ABB RobotStudio station: Task1.rspag

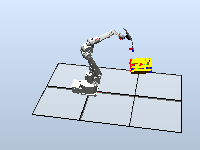
--- station ---
Station t12018 (saved by RobotStudio 6.8.8148.134)
Controller IRB_1520ID_4kg_1.50m
  mechanical unit ROB_1: IRB1520ID_4_150__02, 6 joints, base frame (0, 0, 0) mm
Layout (positions relative to the parent item):
  - IRB1520ID_4_150__02 [mechanism, from Robots\IRB1520ID_4_150_G_02.rslib] at (0, 0, 0) mm; joint values [0.6739, -0.4302, 0.2186, -0.7083, 0.9805, 0.8248] (rad or m)
  - AW_Gun_PSF_25 [mechanism, from Tools\AW_Gun_PSF_25.rslib] at (625.47, 361.2, 1236.61) mm, rotated rx -180 ry 60 rz 180 deg
  - Curve_thing [part, from Training Objects\Curve_Thing.rslib] at (900.38, 149.94, 467.04) mm, rotated rx 0 ry -5.23 rz 7.04 deg
Attachment: AW_Gun_PSF_25 is attached to IRB1520ID_4_150__02 / Link6
Targets, tools, work objects and paths stored in the station and not in the controller backup, written as RAPID:
! task T_ROB1
MODULE Module1
  CONST robtarget Target_50:=[[855.450316917,446.661091818,556.66779203],[0.05059499,0,0.998719253,0],[0,0,0,0],[9E+09,9E+09,9E+09,9E+09,9E+09,9E+09]];
  CONST robtarget Target_240:=[[870.559467167,361.195047252,567.122430983],[0.05059499,0,0.998719253,0],[0,0,0,0],[9E+09,9E+09,9E+09,9E+09,9E+09,9E+09]];
  CONST robtarget Target_60_2:=[[870.559467167,361.195047252,657.122430983],[0.05059499,0,0.998719253,0],[0,0,0,0],[9E+09,9E+09,9E+09,9E+09,9E+09,9E+09]];
  CONST robtarget Target_70_2:=[[888.080268226,219.399873941,657.122430983],[0.05059499,0,0.998719253,0],[0,0,0,0],[9E+09,9E+09,9E+09,9E+09,9E+09,9E+09]];
  CONST robtarget Target_80_2:=[[904.089387296,224.300982937,658.630621291],[0.05059499,0,0.998719253,0],[0,0,0,0],[9E+09,9E+09,9E+09,9E+09,9E+09,9E+09]];
  CONST robtarget Target_90_2:=[[920.816879189,223.596185165,660.141143018],[0.05059499,0,0.998719253,0],[0,0,0,0],[9E+09,9E+09,9E+09,9E+09,9E+09,9E+09]];
  CONST robtarget Target_100_2:=[[936.371952521,217.365147414,661.483254401],[0.05059499,0,0.998719253,0],[0,0,0,0],[9E+09,9E+09,9E+09,9E+09,9E+09,9E+09]];
  CONST robtarget Target_110_2:=[[948.996340197,206.312194788,662.505249932],[0.05059499,0,0.998719253,0],[0,0,0,0],[9E+09,9E+09,9E+09,9E+09,9E+09,9E+09]];
  CONST robtarget Target_120_2:=[[1011.676222413,214.057181596,668.281846254],[0.05059499,0,0.998719253,0],[0,0,0,0],[9E+09,9E+09,9E+09,9E+09,9E+09,9E+09]];
  CONST robtarget Target_130_2:=[[1016.694200617,232.87209655,668.948386567],[0.05059499,0,0.998719253,0],[0,0,0,0],[9E+09,9E+09,9E+09,9E+09,9E+09,9E+09]];
  CONST robtarget Target_140_2:=[[1028.495415861,248.325502176,670.192966537],[0.05059499,0,0.998719253,0],[0,0,0,0],[9E+09,9E+09,9E+09,9E+09,9E+09,9E+09]];
  CONST robtarget Target_150_2:=[[1045.287851693,258.07079632,671.826596493],[0.05059499,0,0.998719253,0],[0,0,0,0],[9E+09,9E+09,9E+09,9E+09,9E+09,9E+09]];
  CONST robtarget Target_160_2:=[[1064.521574005,260.628154485,673.601209461],[0.05059499,0,0.998719253,0],[0,0,0,0],[9E+09,9E+09,9E+09,9E+09,9E+09,9E+09]];
  CONST robtarget Target_170_2:=[[1083.275938942,255.609241416,675.247330174],[0.05059499,0,0.998719253,0],[0,0,0,0],[9E+09,9E+09,9E+09,9E+09,9E+09,9E+09]];
  CONST robtarget Target_180_2:=[[1098.703093142,243.77617988,676.514994934],[0.05059499,0,0.998719253,0],[0,0,0,0],[9E+09,9E+09,9E+09,9E+09,9E+09,9E+09]];
  CONST robtarget Target_190_2:=[[1108.460420734,226.925822191,677.211708641],[0.05059499,0,0.998719253,0],[0,0,0,0],[9E+09,9E+09,9E+09,9E+09,9E+09,9E+09]];
  CONST robtarget Target_200_2:=[[1111.06626994,207.616897902,677.231675207],[0.05059499,0,0.998719253,0],[0,0,0,0],[9E+09,9E+09,9E+09,9E+09,9E+09,9E+09]];
  CONST robtarget Target_210_2:=[[1106.124942133,188.7814703,676.571862704],[0.05059499,0,0.998719253,0],[0,0,0,0],[9E+09,9E+09,9E+09,9E+09,9E+09,9E+09]];
  CONST robtarget Target_220_2:=[[1191.583816693,199.341124094,684.447777639],[0.05059499,0,0.998719253,0],[0,0,0,0],[9E+09,9E+09,9E+09,9E+09,9E+09,9E+09]];
  CONST robtarget Target_230_2:=[[1167.057511069,397.831578102,684.447777639],[0.05059499,0,0.998719253,0],[0,0,0,0],[9E+09,9E+09,9E+09,9E+09,9E+09,9E+09]];
  CONST robtarget Target_10_2:=[[855.450316917,446.661091818,646.66779203],[0.05059499,0,0.998719253,0],[0,0,0,0],[9E+09,9E+09,9E+09,9E+09,9E+09,9E+09]];
  CONST robtarget Target_20_2:=[[892.239775353,148.925410806,646.66779203],[0.05059499,0,0.998719253,0],[0,0,0,0],[9E+09,9E+09,9E+09,9E+09,9E+09,9E+09]];
  CONST robtarget Target_30_2:=[[1287.570500555,197.774118606,683.101587572],[0.05059499,0,0.998719253,0],[0,0,0,0],[9E+09,9E+09,9E+09,9E+09,9E+09,9E+09]];
  CONST robtarget Target_40_2:=[[1250.781042119,495.509799618,683.101587572],[0.05059499,0,0.998719253,0],[0,0,0,0],[9E+09,9E+09,9E+09,9E+09,9E+09,9E+09]];
ENDMODULE


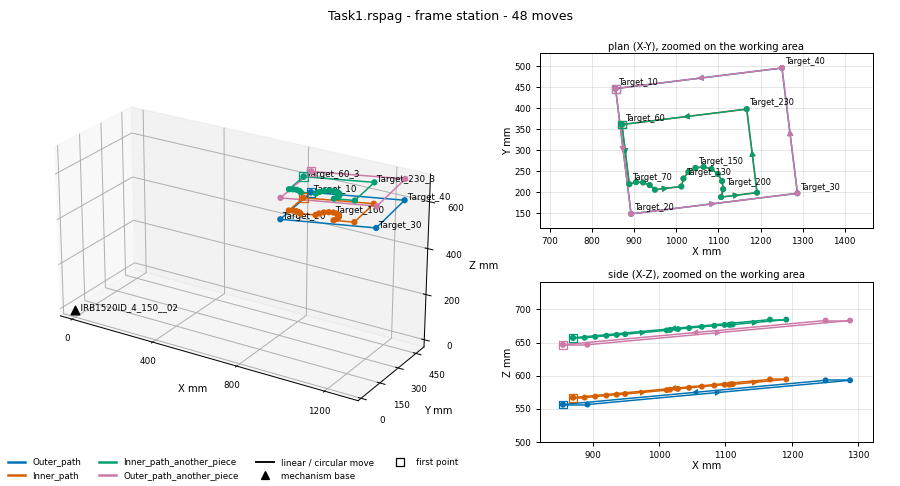
[picture p0: tool path of Task1.rspag in frame station, 48 of 56 moves have a stored position in this frame; points joined in program order, loops and branches not executed]
--- Backups/IRB_1520ID_4kg_1.50m/RAPID/TASK1/PROGMOD/CalibData.mod ---
MODULE CalibData
	PERS tooldata AW_Gun:=[TRUE,[[119.5,0,352],[0.890213743,0,0.455543074,0]],[1,[0,0,100],[1,0,0,0],0,0,0]];
ENDMODULE

--- Backups/IRB_1520ID_4kg_1.50m/RAPID/TASK1/PROGMOD/Module1.mod ---
MODULE Module1
	CONST robtarget Target_10:=[[855.450316917,446.661091818,556.66779203],[0.05059499,0,0.998719253,0],[0,0,0,0],[9E+09,9E+09,9E+09,9E+09,9E+09,9E+09]];
	CONST robtarget Target_20:=[[892.239775353,148.925410806,556.66779203],[0.05059499,0,0.998719253,0],[0,0,0,0],[9E+09,9E+09,9E+09,9E+09,9E+09,9E+09]];
	CONST robtarget Target_30:=[[1287.570500555,197.774118606,593.101587572],[0.05059499,0,0.998719253,0],[0,0,0,0],[9E+09,9E+09,9E+09,9E+09,9E+09,9E+09]];
	CONST robtarget Target_40:=[[1250.781042119,495.509799618,593.101587572],[0.05059499,0,0.998719253,0],[0,0,0,0],[9E+09,9E+09,9E+09,9E+09,9E+09,9E+09]];
	CONST robtarget Target_60:=[[870.559467167,361.195047252,567.122430983],[0.05059499,0,0.998719253,0],[0,0,0,0],[9E+09,9E+09,9E+09,9E+09,9E+09,9E+09]];
	CONST robtarget Target_70:=[[888.080268226,219.399873941,567.122430983],[0.05059499,0,0.998719253,0],[0,0,0,0],[9E+09,9E+09,9E+09,9E+09,9E+09,9E+09]];
	CONST robtarget Target_80:=[[904.089387296,224.300982937,568.630621291],[0.05059499,0,0.998719253,0],[0,0,0,0],[9E+09,9E+09,9E+09,9E+09,9E+09,9E+09]];
	CONST robtarget Target_90:=[[920.816879189,223.596185165,570.141143018],[0.05059499,0,0.998719253,0],[0,0,0,0],[9E+09,9E+09,9E+09,9E+09,9E+09,9E+09]];
	CONST robtarget Target_100:=[[936.371952521,217.365147414,571.483254401],[0.05059499,0,0.998719253,0],[0,0,0,0],[9E+09,9E+09,9E+09,9E+09,9E+09,9E+09]];
	CONST robtarget Target_110:=[[948.996340197,206.312194788,572.505249932],[0.05059499,0,0.998719253,0],[0,0,0,0],[9E+09,9E+09,9E+09,9E+09,9E+09,9E+09]];
	CONST robtarget Target_120:=[[1011.676222413,214.057181596,578.281846254],[0.05059499,0,0.998719253,0],[0,0,0,0],[9E+09,9E+09,9E+09,9E+09,9E+09,9E+09]];
	CONST robtarget Target_130:=[[1016.694200617,232.87209655,578.948386567],[0.05059499,0,0.998719253,0],[0,0,0,0],[9E+09,9E+09,9E+09,9E+09,9E+09,9E+09]];
	CONST robtarget Target_140:=[[1028.495415861,248.325502176,580.192966537],[0.05059499,0,0.998719253,0],[0,0,0,0],[9E+09,9E+09,9E+09,9E+09,9E+09,9E+09]];
	CONST robtarget Target_150:=[[1045.287851693,258.07079632,581.826596493],[0.05059499,0,0.998719253,0],[0,0,0,0],[9E+09,9E+09,9E+09,9E+09,9E+09,9E+09]];
	CONST robtarget Target_160:=[[1064.521574005,260.628154485,583.601209461],[0.05059499,0,0.998719253,0],[0,0,0,0],[9E+09,9E+09,9E+09,9E+09,9E+09,9E+09]];
	CONST robtarget Target_170:=[[1083.275938942,255.609241416,585.247330174],[0.05059499,0,0.998719253,0],[0,0,0,0],[9E+09,9E+09,9E+09,9E+09,9E+09,9E+09]];
	CONST robtarget Target_180:=[[1098.703093142,243.77617988,586.514994934],[0.05059499,0,0.998719253,0],[0,0,0,0],[9E+09,9E+09,9E+09,9E+09,9E+09,9E+09]];
	CONST robtarget Target_190:=[[1108.460420734,226.925822191,587.211708641],[0.05059499,0,0.998719253,0],[0,0,0,0],[9E+09,9E+09,9E+09,9E+09,9E+09,9E+09]];
	CONST robtarget Target_200:=[[1111.06626994,207.616897902,587.231675207],[0.05059499,0,0.998719253,0],[0,0,0,0],[9E+09,9E+09,9E+09,9E+09,9E+09,9E+09]];
	CONST robtarget Target_210:=[[1106.124942133,188.7814703,586.571862704],[0.05059499,0,0.998719253,0],[0,0,0,0],[9E+09,9E+09,9E+09,9E+09,9E+09,9E+09]];
	CONST robtarget Target_220:=[[1191.583816693,199.341124094,594.447777639],[0.05059499,0,0.998719253,0],[0,0,0,0],[9E+09,9E+09,9E+09,9E+09,9E+09,9E+09]];
	CONST robtarget Target_230:=[[1167.057511069,397.831578102,594.447777639],[0.05059499,0,0.998719253,0],[0,0,0,0],[9E+09,9E+09,9E+09,9E+09,9E+09,9E+09]];
    CONST robtarget Target_60_3:=[[870.559467167,361.195047252,657.122430983],[0.05059499,0,0.998719253,0],[0,0,0,0],[9E+09,9E+09,9E+09,9E+09,9E+09,9E+09]];
    CONST robtarget Target_70_3:=[[888.080268226,219.399873941,657.122430983],[0.05059499,0,0.998719253,0],[0,0,0,0],[9E+09,9E+09,9E+09,9E+09,9E+09,9E+09]];
    CONST robtarget Target_80_3:=[[904.089387296,224.300982937,658.630621291],[0.05059499,0,0.998719253,0],[0,0,0,0],[9E+09,9E+09,9E+09,9E+09,9E+09,9E+09]];
    CONST robtarget Target_90_3:=[[920.816879189,223.596185165,660.141143018],[0.05059499,0,0.998719253,0],[0,0,0,0],[9E+09,9E+09,9E+09,9E+09,9E+09,9E+09]];
    CONST robtarget Target_100_3:=[[936.371952521,217.365147414,661.483254401],[0.05059499,0,0.998719253,0],[0,0,0,0],[9E+09,9E+09,9E+09,9E+09,9E+09,9E+09]];
    CONST robtarget Target_110_3:=[[948.996340197,206.312194788,662.505249932],[0.05059499,0,0.998719253,0],[0,0,0,0],[9E+09,9E+09,9E+09,9E+09,9E+09,9E+09]];
    CONST robtarget Target_120_3:=[[1011.676222413,214.057181596,668.281846254],[0.05059499,0,0.998719253,0],[0,0,0,0],[9E+09,9E+09,9E+09,9E+09,9E+09,9E+09]];
    CONST robtarget Target_130_3:=[[1016.694200617,232.87209655,668.948386567],[0.05059499,0,0.998719253,0],[0,0,0,0],[9E+09,9E+09,9E+09,9E+09,9E+09,9E+09]];
    CONST robtarget Target_140_3:=[[1028.495415861,248.325502176,670.192966537],[0.05059499,0,0.998719253,0],[0,0,0,0],[9E+09,9E+09,9E+09,9E+09,9E+09,9E+09]];
    CONST robtarget Target_150_3:=[[1045.287851693,258.07079632,671.826596493],[0.05059499,0,0.998719253,0],[0,0,0,0],[9E+09,9E+09,9E+09,9E+09,9E+09,9E+09]];
    CONST robtarget Target_160_3:=[[1064.521574005,260.628154485,673.601209461],[0.05059499,0,0.998719253,0],[0,0,0,0],[9E+09,9E+09,9E+09,9E+09,9E+09,9E+09]];
    CONST robtarget Target_170_3:=[[1083.275938942,255.609241416,675.247330174],[0.05059499,0,0.998719253,0],[0,0,0,0],[9E+09,9E+09,9E+09,9E+09,9E+09,9E+09]];
    CONST robtarget Target_180_3:=[[1098.703093142,243.77617988,676.514994934],[0.05059499,0,0.998719253,0],[0,0,0,0],[9E+09,9E+09,9E+09,9E+09,9E+09,9E+09]];
    CONST robtarget Target_190_3:=[[1108.460420734,226.925822191,677.211708641],[0.05059499,0,0.998719253,0],[0,0,0,0],[9E+09,9E+09,9E+09,9E+09,9E+09,9E+09]];
    CONST robtarget Target_200_3:=[[1111.06626994,207.616897902,677.231675207],[0.05059499,0,0.998719253,0],[0,0,0,0],[9E+09,9E+09,9E+09,9E+09,9E+09,9E+09]];
    CONST robtarget Target_210_3:=[[1106.124942133,188.7814703,676.571862704],[0.05059499,0,0.998719253,0],[0,0,0,0],[9E+09,9E+09,9E+09,9E+09,9E+09,9E+09]];
    CONST robtarget Target_220_3:=[[1191.583816693,199.341124094,684.447777639],[0.05059499,0,0.998719253,0],[0,0,0,0],[9E+09,9E+09,9E+09,9E+09,9E+09,9E+09]];
    CONST robtarget Target_230_3:=[[1167.057511069,397.831578102,684.447777639],[0.05059499,0,0.998719253,0],[0,0,0,0],[9E+09,9E+09,9E+09,9E+09,9E+09,9E+09]];
    CONST robtarget Target_10_3:=[[855.450316917,446.661091818,646.66779203],[0.05059499,0,0.998719253,0],[0,0,0,0],[9E+09,9E+09,9E+09,9E+09,9E+09,9E+09]];
    CONST robtarget Target_20_3:=[[892.239775353,148.925410806,646.66779203],[0.05059499,0,0.998719253,0],[0,0,0,0],[9E+09,9E+09,9E+09,9E+09,9E+09,9E+09]];
    CONST robtarget Target_30_3:=[[1287.570500555,197.774118606,683.101587572],[0.05059499,0,0.998719253,0],[0,0,0,0],[9E+09,9E+09,9E+09,9E+09,9E+09,9E+09]];
    CONST robtarget Target_40_3:=[[1250.781042119,495.509799618,683.101587572],[0.05059499,0,0.998719253,0],[0,0,0,0],[9E+09,9E+09,9E+09,9E+09,9E+09,9E+09]];
    !***********************************************************
    !
    ! Module:  Module1
    !
    ! Description:
    !   <  Follows a external and a internal part of the given piece
    !       to weld and another workpiece is placed on top of the
    !       workpiece that the robot repeat the welding path >
    !
    ! Author: Khan
    !
    ! Version: 1.0
    !
    !***********************************************************



    PROC main()
        !for 1st workpice
        Outer_path;
        Inner_path;

        WaitTime 3;

        !for another workpice
        Outer_path_another_piece;
        Inner_path_another_piece;


    ENDPROC

	PROC Outer_path()

        VAR robtarget vertical_point; !declearing variable for offset
        vertical_point:=Offs(Target_10, 0, 0, 300); !creating the offset 300mm above of the starting point

        MoveL vertical_point,v500,z0,AW_Gun\WObj:=wobj0; !as the welding should be precise, z0 is taken for every terget
	    MoveL Target_10,v500,z0,AW_Gun\WObj:=wobj0; !welding start point
	    MoveL Target_20,v500,z0,AW_Gun\WObj:=wobj0;
	    MoveL Target_30,v500,z0,AW_Gun\WObj:=wobj0;
	    MoveL Target_40,v500,z0,AW_Gun\WObj:=wobj0;
	    MoveL Target_10,v500,z0,AW_Gun\WObj:=wobj0; !welding end point
        MoveL vertical_point,v500,z0,AW_Gun\WObj:=wobj0;
	ENDPROC

	PROC Inner_path()

        VAR robtarget vertical_point; !declearing variable for offset
        vertical_point:=Offs(Target_60, 0, 0, 300); !creating the offset 300mm above of the starting point

        MoveL vertical_point,v500,z0,AW_Gun\WObj:=wobj0;!as the welding should be precise, z0 is taken for every terget
	    MoveL Target_60,v500,z0,AW_Gun\WObj:=wobj0; !welding start point
	    MoveL Target_70,v500,z0,AW_Gun\WObj:=wobj0;
	    MoveL Target_80,v500,z0,AW_Gun\WObj:=wobj0;
	    MoveL Target_90,v500,z0,AW_Gun\WObj:=wobj0;
	    MoveL Target_100,v500,z0,AW_Gun\WObj:=wobj0;
	    MoveL Target_110,v500,z0,AW_Gun\WObj:=wobj0;
	    MoveL Target_120,v500,z0,AW_Gun\WObj:=wobj0;
	    MoveL Target_130,v500,z0,AW_Gun\WObj:=wobj0;
	    MoveL Target_140,v500,z0,AW_Gun\WObj:=wobj0;
	    MoveL Target_150,v500,z0,AW_Gun\WObj:=wobj0;
	    MoveL Target_160,v500,z0,AW_Gun\WObj:=wobj0;
	    MoveL Target_170,v500,z0,AW_Gun\WObj:=wobj0;
	    MoveL Target_180,v500,z0,AW_Gun\WObj:=wobj0;
	    MoveL Target_190,v500,z0,AW_Gun\WObj:=wobj0;
	    MoveL Target_200,v500,z0,AW_Gun\WObj:=wobj0;
	    MoveL Target_210,v500,z0,AW_Gun\WObj:=wobj0;
	    MoveL Target_220,v500,z0,AW_Gun\WObj:=wobj0;
	    MoveL Target_230,v500,z0,AW_Gun\WObj:=wobj0;
	    MoveL Target_60,v500,z0,AW_Gun\WObj:=wobj0; !welding end point
        MoveL vertical_point,v500,z0,AW_Gun\WObj:=wobj0;
	ENDPROC


    PROC Inner_path_another_piece()

        VAR robtarget vertical_point;
        vertical_point:=Offs(Target_60_3, 0, 0, 300);

        MoveL vertical_point,v500,z0,AW_Gun\WObj:=wobj0;
        MoveL Target_60_3,v500,z0,AW_Gun\WObj:=wobj0; !welding start point
        MoveL Target_70_3,v500,z0,AW_Gun\WObj:=wobj0;
        MoveL Target_80_3,v500,z0,AW_Gun\WObj:=wobj0;
        MoveL Target_90_3,v500,z0,AW_Gun\WObj:=wobj0;
        MoveL Target_100_3,v500,z0,AW_Gun\WObj:=wobj0;
        MoveL Target_110_3,v500,z0,AW_Gun\WObj:=wobj0;
        MoveL Target_120_3,v500,z0,AW_Gun\WObj:=wobj0;
        MoveL Target_130_3,v500,z0,AW_Gun\WObj:=wobj0;
        MoveL Target_140_3,v500,z0,AW_Gun\WObj:=wobj0;
        MoveL Target_150_3,v500,z0,AW_Gun\WObj:=wobj0;
        MoveL Target_160_3,v500,z0,AW_Gun\WObj:=wobj0;
        MoveL Target_170_3,v500,z0,AW_Gun\WObj:=wobj0;
        MoveL Target_180_3,v500,z0,AW_Gun\WObj:=wobj0;
        MoveL Target_190_3,v500,z0,AW_Gun\WObj:=wobj0;
        MoveL Target_200_3,v500,z0,AW_Gun\WObj:=wobj0;
        MoveL Target_210_3,v500,z0,AW_Gun\WObj:=wobj0;
        MoveL Target_220_3,v500,z0,AW_Gun\WObj:=wobj0;
        MoveL Target_230_3,v500,z0,AW_Gun\WObj:=wobj0;
        MoveL Target_60_3,v500,z0,AW_Gun\WObj:=wobj0; !welding end point
        MoveL vertical_point,v500,z0,AW_Gun\WObj:=wobj0;
        ENDPROC

    PROC Outer_path_another_piece()

        VAR robtarget vertical_point;
        vertical_point:=Offs(Target_10_3, 0, 0, 300);

        MoveL vertical_point,v500,z0,AW_Gun\WObj:=wobj0;
        MoveL Target_10_3,v500,z0,AW_Gun\WObj:=wobj0; !welding start point
        MoveL Target_20_3,v500,z0,AW_Gun\WObj:=wobj0;
        MoveL Target_30_3,v500,z0,AW_Gun\WObj:=wobj0;
        MoveL Target_40_3,v500,z0,AW_Gun\WObj:=wobj0;
        MoveL Target_10_3,v500,z0,AW_Gun\WObj:=wobj0; !welding end point
        MoveL vertical_point,v500,z0,AW_Gun\WObj:=wobj0;
    ENDPROC
ENDMODULE
